// TIA Portal V19 export
TYPE "LUC_typeStateConfiguration"
// Configure which states are enabled for each mode
// stored: Access Published
   STRUCT
      clearing : Bool := true;   // Enable state Clearing
      starting : Bool := true;   // Enable state Starting
      suspended : Bool := true;   // Enable state Suspended
      stopping : Bool := true;   // Enable state Stopping
      aborting : Bool := true;   // Enable state Aborting
      holding : Bool := true;   // Enable state Holding
      held : Bool := true;   // Enable state Held
      unholding : Bool := true;   // Enable state Unholding
      suspending : Bool := true;   // Enable state Suspending
      unsuspending : Bool := true;   // Enable state Unsuspending
      resetting : Bool := true;   // Enable state Resetting
      completing : Bool := true;   // Enable state Completing
      completed : Bool := true;   // Enable state Completed
   END_STRUCT;
END_TYPE
